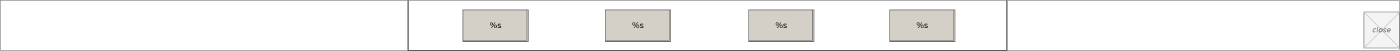
VISUALIZATION VISU_BANDEAU_CFG  // 1916x70, background image fond ecran
    Rectangle (558,0 820x70)
    Image (1866,16 50x50), image: close
        tap Global_Variables.RQ_PARAM_SYSTEM
        OnMouseClick: toggle RQ_PARAM_SYSTEM
        OnMouseClick: change screen: SYN_PROC
    Button (633,13 90x44), "%s", text list: 'TextList_Navigation', text index: 3
        OnMouseClick: change screen: VISU_CONFIG_POMPAGE
    Button (1217,13 90x44), "%s", text list: 'TextList_Navigation', text index: 4
        OnMouseClick: change screen: VISU_CONFIG_EVAP
    Button (828,13 90x44), "%s", text list: 'TextList_Navigation', text index: 8
        OnMouseClick: change screen: VISU_CONFIG_GAZ
    Button (1024,13 90x44), "%s", text list: 'TextList_Navigation', text index: 13
        OnMouseClick: change screen: VISU_CONFIG_REGEN
END_VISUALIZATION

(* stored: Version 1.1.0.1, ProductVersion 3.1.4026.18
   Visu VISU_BANDEAU_CFG: Id {13778180-60c5-4262-bfa7-c1669fc8a06c} *)
